TYPE ST_Axis :
STRUCT
	IN	: ST_AxisIn;
	OUT	: ST_AxisOut;
	
END_STRUCT
END_TYPE

(* stored: Version 1.1.0.1, ProductVersion 3.1.4022.12
   DUT ST_Axis: Id {5465b3b0-c2de-4b12-b512-7c7e24913e6d} *)
